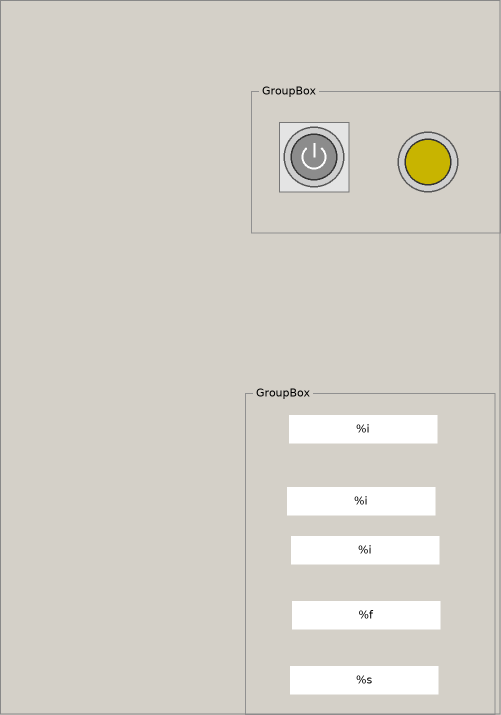
VISUALIZATION HMI  // 501x715
    GroupBox (251,83 250x150), "GroupBox"
        PowerSwitch (28,39 70x70), variable: MAIN.bStart, behaviour: TOGGLE, style: Switch-PowerSwitch-Gray
        Lamp1 (142,44 70x70), variable: MAIN.bStart, style: Lamp-Lamp1-Yellow
    GroupBox (245,385 250x330), "GroupBox"
        Textfield (45,150 150x30), "%i", text variable: MAIN.nUINT
        Textfield (46,215 150x30), "%f", text variable: MAIN.fREAL
        Textfield (43,29 150x30), "%i", text variable: Main.bEnable
        Textfield (44,280 150x30), "%s", text variable: MAIN.sPowerStatus
        Textfield (41,101 150x30), "%i", text variable: MAIN.nINT
END_VISUALIZATION

(* stored: Version 1.1.0.1, ProductVersion 3.1.4024.12
   Visu HMI: Id {da3deb83-6604-4901-a11f-ac5a3b78a6e8} *)
